FUNCTION_BLOCK FB_Room

VAR
	 sOutput : STRING := '';
END_VAR

METHOD FB_init : BOOL
VAR_INPUT
	bInitRetains : BOOL; // if TRUE, the retain variables are initialized (warm start / cold start)
	bInCopyCode : BOOL;  // if TRUE, the instance afterwards gets moved into the copy code (online change)
END_VAR
sOutput := 'Room created inside House';
END_METHOD

END_FUNCTION_BLOCK

(* stored: Version 1.1.0.1, ProductVersion 3.1.4024.16
   POU FB_Room: Id {c99913c1-4235-4642-acb7-c51c880677d5}, SpecialFunc None
   Method FB_init: Id {2f52d198-f209-4226-8da2-38864d17eea6} *)
